// TIA Portal V18 export
FUNCTION_BLOCK "Timers"   // FB21, LAD
TITLE = Timers
{ S7_Optimized_Access := 'TRUE' }
// Written By Kristopher Gimenez March 3rd,2023
// 
// This block and its DB will contain the system runtimes logic and data
// stored: AutoNumber false, MemoryReserve 100, SetENOAutomatically false
   VAR
      TDTimeReset : Bool;   // Bit set from HMI used to reset time
      M1TimeReset : Bool;   // Bit set from HMI used to reset time
      M2TimeReset : Bool;   // Bit set from HMI used to reset time
      AuxTimeReset : Bool;   // Bit set from HMI used to reset time
      CoolerTimeReset : Bool;   // Bit set from HMI used to reset time
      TDRuntime : "Runtime_Out";
      M1Runtime { S7_SetPoint := 'True'} : "Runtime_Out";
      M2Runtime { S7_SetPoint := 'True'} : "Runtime_Out";
      AuxRuntime { S7_SetPoint := 'True'} : "Runtime_Out";
      CoolerRuntime { S7_SetPoint := 'True'} : "Runtime_Out";
      SystemRunStart : Bool;
      System_Runtime { S7_SetPoint := 'True'} : "Runtime";
      M1_Runtime { S7_SetPoint := 'True'} : "Runtime";
      M2_Runtime { S7_SetPoint := 'True'} : "Runtime";
      Cooler_Runtime { S7_SetPoint := 'True'} : "Runtime";
      AuxPump_Runtime { S7_SetPoint := 'True'} : "Runtime";
   END_VAR
BEGIN

REGION Network 1: TD Run Time
   // Call Each cycle. Reset from HMI
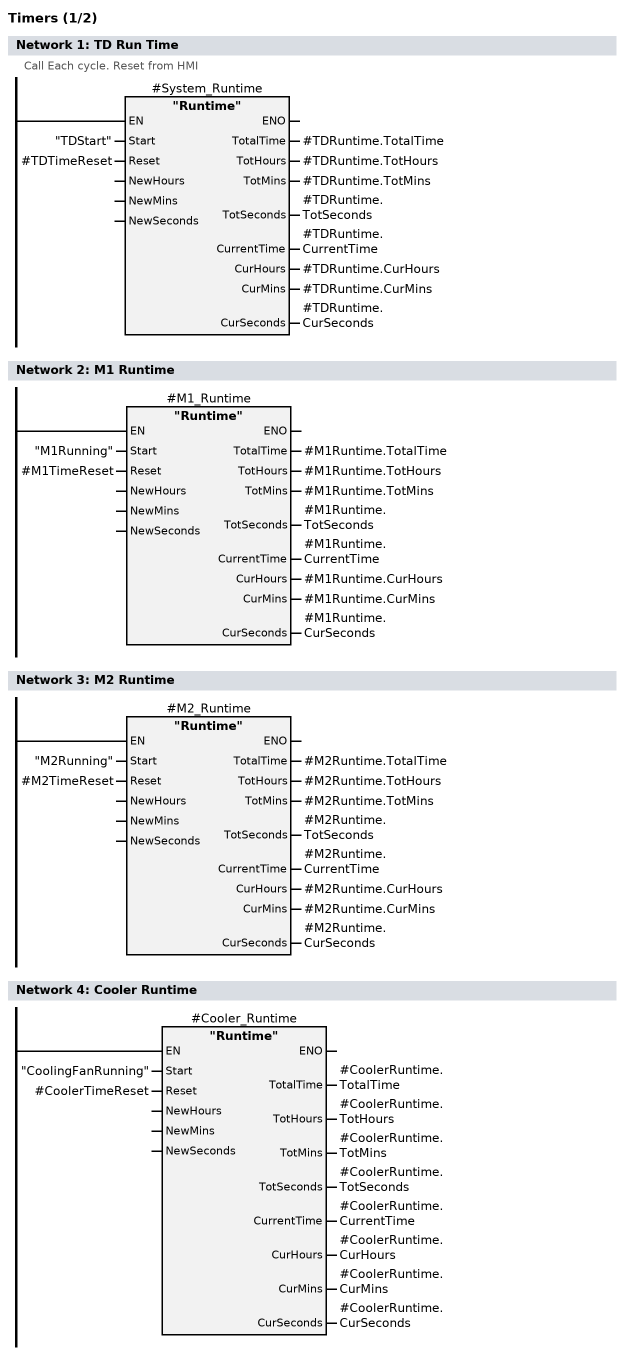
   RUNG wire#powerrail
      #System_Runtime(Start := "TDStart", Reset := #TDTimeReset, NewHours :=, NewMins :=, NewSeconds :=, TotalTime => #TDRuntime.TotalTime, TotHours => #TDRuntime.TotHours, TotMins => #TDRuntime.TotMins, TotSeconds => #TDRuntime.TotSeconds, CurrentTime => #TDRuntime.CurrentTime, CurHours => #TDRuntime.CurHours, CurMins => #TDRuntime.CurMins, CurSeconds => #TDRuntime.CurSeconds)
   END_RUNG
   // the same network as SCL:
   #System_Runtime(Start := "TDStart",   // "Runtime"
                   Reset := #TDTimeReset,
                   TotalTime => #TDRuntime.TotalTime,
                   TotHours => #TDRuntime.TotHours,
                   TotMins => #TDRuntime.TotMins,
                   TotSeconds => #TDRuntime.TotSeconds,
                   CurrentTime => #TDRuntime.CurrentTime,
                   CurHours => #TDRuntime.CurHours,
                   CurMins => #TDRuntime.CurMins,
                   CurSeconds => #TDRuntime.CurSeconds);
END_REGION

REGION Network 2: M1 Runtime
   RUNG wire#powerrail
      #M1_Runtime(Start := "M1Running", Reset := #M1TimeReset, NewHours :=, NewMins :=, NewSeconds :=, TotalTime => #M1Runtime.TotalTime, TotHours => #M1Runtime.TotHours, TotMins => #M1Runtime.TotMins, TotSeconds => #M1Runtime.TotSeconds, CurrentTime => #M1Runtime.CurrentTime, CurHours => #M1Runtime.CurHours, CurMins => #M1Runtime.CurMins, CurSeconds => #M1Runtime.CurSeconds)
   END_RUNG
   // the same network as SCL:
   #M1_Runtime(Start := "M1Running",   // "Runtime"
               Reset := #M1TimeReset,
               TotalTime => #M1Runtime.TotalTime,
               TotHours => #M1Runtime.TotHours,
               TotMins => #M1Runtime.TotMins,
               TotSeconds => #M1Runtime.TotSeconds,
               CurrentTime => #M1Runtime.CurrentTime,
               CurHours => #M1Runtime.CurHours,
               CurMins => #M1Runtime.CurMins,
               CurSeconds => #M1Runtime.CurSeconds);
END_REGION

REGION Network 3: M2 Runtime
   RUNG wire#powerrail
      #M2_Runtime(Start := "M2Running", Reset := #M2TimeReset, NewHours :=, NewMins :=, NewSeconds :=, TotalTime => #M2Runtime.TotalTime, TotHours => #M2Runtime.TotHours, TotMins => #M2Runtime.TotMins, TotSeconds => #M2Runtime.TotSeconds, CurrentTime => #M2Runtime.CurrentTime, CurHours => #M2Runtime.CurHours, CurMins => #M2Runtime.CurMins, CurSeconds => #M2Runtime.CurSeconds)
   END_RUNG
   // the same network as SCL:
   #M2_Runtime(Start := "M2Running",   // "Runtime"
               Reset := #M2TimeReset,
               TotalTime => #M2Runtime.TotalTime,
               TotHours => #M2Runtime.TotHours,
               TotMins => #M2Runtime.TotMins,
               TotSeconds => #M2Runtime.TotSeconds,
               CurrentTime => #M2Runtime.CurrentTime,
               CurHours => #M2Runtime.CurHours,
               CurMins => #M2Runtime.CurMins,
               CurSeconds => #M2Runtime.CurSeconds);
END_REGION

REGION Network 4: Cooler Runtime
   RUNG wire#powerrail
      #Cooler_Runtime(Start := "CoolingFanRunning", Reset := #CoolerTimeReset, NewHours :=, NewMins :=, NewSeconds :=, TotalTime => #CoolerRuntime.TotalTime, TotHours => #CoolerRuntime.TotHours, TotMins => #CoolerRuntime.TotMins, TotSeconds => #CoolerRuntime.TotSeconds, CurrentTime => #CoolerRuntime.CurrentTime, CurHours => #CoolerRuntime.CurHours, CurMins => #CoolerRuntime.CurMins, CurSeconds => #CoolerRuntime.CurSeconds)
   END_RUNG
   // the same network as SCL:
   #Cooler_Runtime(Start := "CoolingFanRunning",   // "Runtime"
                   Reset := #CoolerTimeReset,
                   TotalTime => #CoolerRuntime.TotalTime,
                   TotHours => #CoolerRuntime.TotHours,
                   TotMins => #CoolerRuntime.TotMins,
                   TotSeconds => #CoolerRuntime.TotSeconds,
                   CurrentTime => #CoolerRuntime.CurrentTime,
                   CurHours => #CoolerRuntime.CurHours,
                   CurMins => #CoolerRuntime.CurMins,
                   CurSeconds => #CoolerRuntime.CurSeconds);
END_REGION

REGION Network 5: Aux Pump Runtime
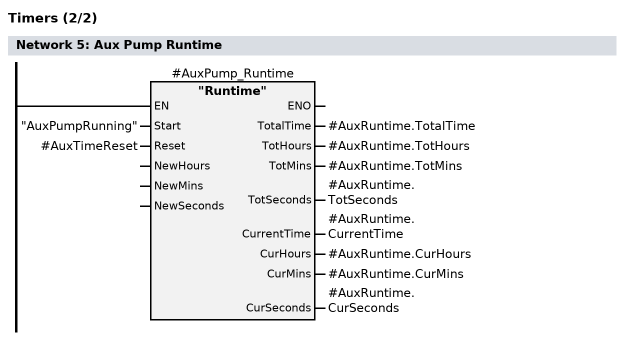
   RUNG wire#powerrail
      #AuxPump_Runtime(Start := "AuxPumpRunning", Reset := #AuxTimeReset, NewHours :=, NewMins :=, NewSeconds :=, TotalTime => #AuxRuntime.TotalTime, TotHours => #AuxRuntime.TotHours, TotMins => #AuxRuntime.TotMins, TotSeconds => #AuxRuntime.TotSeconds, CurrentTime => #AuxRuntime.CurrentTime, CurHours => #AuxRuntime.CurHours, CurMins => #AuxRuntime.CurMins, CurSeconds => #AuxRuntime.CurSeconds)
   END_RUNG
   // the same network as SCL:
   #AuxPump_Runtime(Start := "AuxPumpRunning",   // "Runtime"
                    Reset := #AuxTimeReset,
                    TotalTime => #AuxRuntime.TotalTime,
                    TotHours => #AuxRuntime.TotHours,
                    TotMins => #AuxRuntime.TotMins,
                    TotSeconds => #AuxRuntime.TotSeconds,
                    CurrentTime => #AuxRuntime.CurrentTime,
                    CurHours => #AuxRuntime.CurHours,
                    CurMins => #AuxRuntime.CurMins,
                    CurSeconds => #AuxRuntime.CurSeconds);
END_REGION
END_FUNCTION_BLOCK
